{attribute addProperty BoxType "EL3161-0000-0018"}
{attribute addProperty Id "AI_StandardAT %I*AI_Standard_087F71C73240WcStateAT %I*WcState_F855686C1620InfoDataAT %I*InfoData_BC63D37F80100"}
{attribute addProperty CRC "1089245502"}
{attribute addProperty SizeInBites "128"}
{attribute addProperty SizeInBytes "16"}
TYPE EL3161_60464DCF :
STRUCT
	{attribute addProperty Name "AI_Standard"}
	AI_Standard : AI_Standard_087F71C7;
	{attribute addProperty Name "WcState"}
	WcState : WcState_F855686C;
	{attribute addProperty Name "InfoData"}
	InfoData : InfoData_BC63D37F;
END_STRUCT
END_TYPE

(* stored: Version 1.2.0.0, ProductVersion 3.1.4024.9
   DUT EL3161_60464DCF: Id {9f655c38-81f5-4fc0-a23a-16f9f803d244} *)
